FUNCTION_BLOCK FB_MoveLinear
VAR_INPUT
END_VAR
VAR_OUTPUT
END_VAR
VAR
END_VAR

END_FUNCTION_BLOCK

(* stored: Version 1.1.0.1, ProductVersion 3.1.4022.18
   POU FB_MoveLinear: Id {3e372f47-4d87-428e-8b42-a4cd3e7b0d3b}, SpecialFunc None *)
